// TIA Portal V19 export
DATA_BLOCK "Itf"   // DB1
{ S7_Optimized_Access := 'TRUE' }
// stored: MemoryReserve 0
   VAR
      prendi : Bool;
      posa : Bool;
      accendiAsse : Bool;
      vaiAHomeAsse : Bool;
      pinzaAperta : Bool;
      pinzaChiusa : Bool;
      inPosAlta : Bool;
      inPosBassa : Bool;
      asseAcceso : Bool;
      asseReferenziato : Bool;
      errori : Bool;
      fineMissionePresa : Bool;
      fineMissionePosa : Bool;
      posizioneAttuale : Real;
   END_VAR
BEGIN
END_DATA_BLOCK
